// TIA Portal project "WinCC_Analog_Learn" (V15.1)
// En este proyecto se configura un app en wincc para controlar el variador de velocidad con el DAC del s7-1200.

(* hardware
DEVICE "S7-1200 station_1"  S7-1200 Station
   slot 0: "Rack_0"  S7-1200 Rack  Rack  V1.0
   slot 1: "PLC_1"  CPU 1214C AC/DC/Rly  6ES7 214-1BG40-0XB0  V4.2
   slot 3: "AQ 1x12BIT_1"  AQ1 signal board  6ES7 232-4HA30-0XB0  V1.0
DEVICE "PC-System_1"  SIMATIC PC station
   slot 0: "Estación PC SIMATIC"  Rail  SIMATIC PC-Station  V1.0
      slot 125: "Stationmanager"  Station_Manager  V6.0.4
   slot 1: "HMI_RT_1"  WinCC RT Advanced  6AV2 104-0xxxx-xxxx  15.1.0.0
      slot 33792: "Interfaz host"  Host interface
   slot 2: "IE general_1"  IE General  IE_CP  V8.2.0
*)

// ===== PLC "PLC_1"  CPU 1214C AC/DC/Rly =====

VAR_GLOBAL   // PLC tag table "Tabla de variables estándar"
   "On_Off_Q" AT %M0.0 : Bool;
   "SalidaTest" AT %Q0.0 : Bool;
   "WinCCAnalogVar" AT %MD50 : DWord;
   "NormalizedVal" AT %MD60 : Real;
   "DAC" AT %QW80 : Int;
   "varTest" AT %MW100 : Int;
   "Tag_1" AT %MD120 : DWord;
END_VAR

ORGANIZATION_BLOCK "Main"   // OB1, LAD, ProgramCycle
TITLE = "Main Program Sweep (Cycle)"
{ S7_Optimized_Access := 'TRUE' }
VERSION : 0.1
   VAR_INPUT
      Initial_Call : Bool;   // Initial call of this OB
      Remanence : Bool;   // =True, if remanent data are available
   END_VAR
BEGIN

REGION Network 1
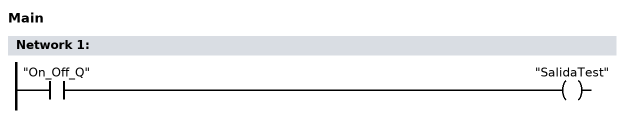
   RUNG wire#powerrail
      Contact( "On_Off_Q" )
      Coil( "SalidaTest" )
   END_RUNG
   // the same network as SCL:
   "SalidaTest" := "On_Off_Q";
END_REGION
END_ORGANIZATION_BLOCK

(* ===== HMI "HMI_RT_1" =====
system functions are stored by id; their names below are inferred from use
connection "HMI_Conexión_1": ETHERNET, S7_1200_OMS

HMI tags "Tabla de variables estándar"
   "On_Off_Q" : Bool = PLC On_Off_Q AT %M0.0, 1 s
   "DAC" : Int = PLC DAC AT %QW80, 1 s
   "varTest" : Int = PLC varTest AT %MW100, 1 s
   "WinCCAnalogVar" : DWord = PLC WinCCAnalogVar AT %MD50, 1 s

screen "Imagen_1" 600x800
   Button "Botón_1" at 47,195 size 137x39; TextOff 'm0.0'
      on Press: InvertBit("On_Off_Q")
   TextField "Campo de texto_1" at 62,263 size 133x22; Text 'Salida Analogica'
   TextField "Campo de texto_2" at 34,157 size 251x22; Text 'Alternar Q0.0 (TEST CONEXION)'
   Slider "Deslizador_1" at 159,294 size 60x377; Caption 'DAC - QW80'
      ProcessValue <- "DAC"
   TextField "Campo de texto_3" at 232,649 size 15x22; Text '0'
   TextField "Campo de texto_4" at 232,477 size 15x22; Text '5'
   TextField "Campo de texto_5" at 232,313 size 25x22; Text '10'
*)